{attribute 'call_after_init'}
FUNCTION_BLOCK FB_AmphosEnable_Test EXTENDS FB_TestSuite
VAR_INPUT
END_VAR
VAR_OUTPUT
END_VAR
VAR
END_VAR

LocksWithHardwareFailure();
EnablesWithAmphosMinorError();
LocksWithAmphosCriticalError();
EnablesWhenNoError();
LocksWithPrevError();
UnlocksWithBeamErrorReset();

METHOD EnablesWhenNoError
VAR
	stErrors : st_ErrorStates;
	stAmphosSetpoints : ST_LaserSetpoints := F_LaserSetpoints();
	bResult : BOOL;
END_VAR
TEST('EnablesWhenNoError');

bResult := F_AmphosEnable(
	fAmphosVoltage := stAmphosSetpoints.nMinNominalVoltage,
	bEnabled := TRUE,
	stAmphosSetpoints := stAmphosSetpoints,
	stErrors := stErrors
);
AssertTrue(bResult, 'Amphos did not enable');

TEST_FINISHED();
END_METHOD

METHOD EnablesWithAmphosMinorError
VAR
	stErrors : st_ErrorStates;
	stAmphosSetpoints : ST_LaserSetpoints := F_LaserSetpoints();
	bResult : BOOL;
END_VAR
TEST('EnablesWithAmphosMinorError');

stErrors.bAmphosBeam := TRUE;
bResult := F_AmphosEnable(
	fAmphosVoltage := stAmphosSetpoints.nMinNominalVoltage - 0.001,
	bEnabled := TRUE,
	stAmphosSetpoints := stAmphosSetpoints,
	stErrors := stErrors
);
AssertTrue(bResult, 'Amphos did not enable');

TEST_FINISHED();
END_METHOD

METHOD LocksWithAmphosCriticalError
VAR
	stErrors : st_ErrorStates;
	stAmphosSetpoints : ST_LaserSetpoints := F_LaserSetpoints();
	bResult : BOOL;
END_VAR
TEST('LocksWithAmphosCriticalError');

stErrors.bAmphosBeam := TRUE;
bResult := F_AmphosEnable(
	fAmphosVoltage := stAmphosSetpoints.nMinVoltage - 0.1,
	bEnabled := TRUE,
	stAmphosSetpoints := stAmphosSetpoints,
	stErrors := stErrors
);
AssertFalse(bResult, 'Amphos did not lock');

TEST_FINISHED();
END_METHOD

METHOD LocksWithHardwareFailure
VAR
	stErrors : st_ErrorStates;
	stAmphosSetpoints : ST_LaserSetpoints := F_LaserSetpoints();
	bResult : BOOL;
END_VAR
TEST('LocksWithHardwareFailure');

stErrors.bHardwareFailure := TRUE;
bResult := F_AmphosEnable(
	fAmphosVoltage := stAmphosSetpoints.nMinNominalVoltage,
	bEnabled := TRUE,
	stAmphosSetpoints := stAmphosSetpoints,
	stErrors := stErrors
);
AssertFalse(bResult, 'Amphos did not lock');

TEST_FINISHED();
END_METHOD

METHOD LocksWithPrevError
VAR
	stErrors : st_ErrorStates;
	stAmphosSetpoints : ST_LaserSetpoints := F_LaserSetpoints();
	bResult : BOOL;
END_VAR
TEST('LatchesWithAmphosCriticalError');

// If the interlock previously failed and there is still a beam error, then lock and stay locked until beam error reset, even if there is only a minor error
stErrors.bAmphosBeam := TRUE;
bResult := F_AmphosEnable(
	fAmphosVoltage := stAmphosSetpoints.nMinNominalVoltage - 0.001, // Minor error
	bEnabled := FALSE,
	stAmphosSetpoints := stAmphosSetpoints,
	stErrors := stErrors
);
AssertFalse(bResult, 'Amphos did not lock');

TEST_FINISHED();
END_METHOD

METHOD UnlocksWithBeamErrorReset
VAR
	stErrors : st_ErrorStates;
	stAmphosSetpoints : ST_LaserSetpoints := F_LaserSetpoints();
	bResult : BOOL;
END_VAR
TEST('Unlocks with beam error reset');

// Even if bEnabled was false last time, reset if the beam error is now cleared
bResult := F_AmphosEnable(
	fAmphosVoltage := stAmphosSetpoints.nMinNominalVoltage,
	bEnabled := FALSE,
	stAmphosSetpoints := stAmphosSetpoints,
	stErrors := stErrors
);
AssertTrue(bResult, 'Amphos did not enable');

TEST_FINISHED();
END_METHOD

END_FUNCTION_BLOCK

(* stored: Version 1.1.0.1, ProductVersion 3.1.4020.14
   POU FB_AmphosEnable_Test: Id {c0048a71-40cb-425a-920b-fa92fa66b08c}, SpecialFunc None
   Method EnablesWhenNoError: Id {78be0b16-fc82-4ade-a9ba-17eb954ac394}
   Method EnablesWithAmphosMinorError: Id {a96a87a0-02d5-47d7-bd7b-8eb1f93767db}
   Method LocksWithAmphosCriticalError: Id {eab64e8c-fe99-4322-be86-62443c42d485}
   Method LocksWithHardwareFailure: Id {ea342f1c-19f4-449a-ac36-8ddd6bb1a06e}
   Method LocksWithPrevError: Id {eabe7bf9-7626-468b-a342-db7c28449f22}
   Method UnlocksWithBeamErrorReset: Id {12874555-36bd-41ee-9054-354d4c598132} *)
